FUNCTION_BLOCK SignalTimeComparison
VAR_INPUT
	insignalTime	:	ULINT;
	outsignalTime	:	ULINT;
END_VAR
VAR_OUTPUT
	seconds	:	ULINT;
	milseconds	:	ULINT;
	micseconds	:	ULINT;
	nseconds	:	ULINT;
END_VAR
VAR
END_VAR
VAR CONSTANT
	noOfSamples	:	INT := 19;
END_VAR

nseconds := (insignalTime MOD 1000) - (outsignalTime MOD 1000);

micseconds := ((insignalTime MOD 1000000) - (outsignalTime MOD 1000000))/1000;

milseconds := ((insignalTime MOD 1000000000) - (outsignalTime MOD 1000000000))/1000000;

seconds := (insignalTime/1000000000) - (outsignalTime/1000000000);

END_FUNCTION_BLOCK

(* stored: Version 1.1.0.1, ProductVersion 3.1.4024.12
   POU SignalTimeComparison: Id {2d963246-5fc1-4831-ad2c-9f109bc44b9c}, SpecialFunc None *)
